{attribute 'no_check'}
FUNCTION_BLOCK IOMotor IMPLEMENTS I_ActuatorOnOff
VAR_INPUT
	ResetTrig												:	BOOL := TRUE; //Confirm error
	start													:	BOOL;
	Feed													:	BOOL;
	ProtSwitchOK											: 	FUSE;
END_VAR                 							
VAR_OUTPUT
{attribute 'displaymode':='binary'}
	Status													:	BYTE;              							
	Q_Contactor										AT  %Q* :	BOOL; //Hardware output for main contactor to start motor	
	Busy													:	BOOL;
	Error													:	BOOL;
END_VAR                 							
VAR (* IO Internal *)   							

                        	
END_VAR                 	
VAR                     	
END_VAR

(* Com Motor IO 					 		V2.2		*)
(********************************************************)

(* Protection Switch *****************************************)
	IF ResetTrig THEN reset(); END_IF

	ProtSwitchOK();

(* Enable ****************************************************)
	IF Start THEN
		switchOn();
	ELSE
		switchOff();
	END_IF
	
(* HMI status *********************************************)
	_writeStatus();
	
(********************************************************)

METHOD PROTECTED _writeStatus : BOOL
VAR_INPUT
END_VAR
	
(* HmiStatus **************************************************)
	Status.0												:= NOT Q_Contactor;
	Status.1												:= Q_Contactor;
	Status.2												:= FALSE;
	Status.3												:= FALSE;
	Status.4												:= FALSE;
	Status.5												:= Feed ;
	Status.6												:= NOT Error;
	Status.7												:= Error;

	(* Result *)
	_writeStatus											:= TRUE;
    												
(**************************************************************)
END_METHOD

METHOD enable : BOOL //Result value = successful execution of desired action 
VAR_INPUT
	IN							:	BOOL; //TRUE = Enable Pos/FWD/Up/Open/Left/Work FALSE = Opposite
END_VAR
IF in
THEN
	enable := switchOn();
ELSE
	enable := switchOff();
END_IF
END_METHOD

{attribute 'monitoring' := 'call'}
PROPERTY public inError : bool
GET
inError := Error;
END_GET
END_PROPERTY

{attribute 'monitoring' := 'call'}
PROPERTY public isBusy : bool
GET
isBusy := Busy;
END_GET
END_PROPERTY

{attribute 'monitoring' := 'call'}
PROPERTY public isOff : BOOL
GET
isOff := not Q_Contactor;
END_GET
END_PROPERTY

{attribute 'monitoring' := 'call'}
PROPERTY public isOn : BOOL
GET
isOn := Q_Contactor;
END_GET
END_PROPERTY

{attribute 'monitoring' := 'call'}
PROPERTY noFeed : BOOL
GET
noFeed := NOT Feed;
END_GET
END_PROPERTY

{attribute 'monitoring' := 'call'}
PROPERTY ok : bool
GET
ok := isBusy;
END_GET
END_PROPERTY

METHOD PUBLIC reset : bool
VAR_INPUT
END_VAR
Error									:= FALSE;
reset									:= ProtSwitchOK.reset();
END_METHOD

METHOD public switchOff : BOOL  //True if motor is switched off
VAR_INPUT
END_VAR
Start														:= FALSE;
Q_Contactor 												:= FALSE;
Busy														:= FALSE;
Error														:= NOT ProtSwitchOK.Q;
switchOff													:= TRUE;
END_METHOD

METHOD public switchOn : BOOL  //True if motor is switched on
VAR_INPUT
END_VAR
Start														:= TRUE;
Q_Contactor		 											:= ProtSwitchOK.Q AND Feed;
switchOn													:= Q_Contactor;
Busy														:= switchOn;
Error														:= NOT ProtSwitchOK.Q;
END_METHOD

END_FUNCTION_BLOCK

(* stored: Version 1.1.0.1, ProductVersion 3.1.4024.3
   POU IOMotor: Id {652201da-3ead-4c30-bab1-0ca4c35805c5}, SpecialFunc None
   Folder methods: Id {279f1738-11a0-4557-bc76-03636caa0103}
   Folder properties: Id {cdc3a8c6-d9ab-45f4-9e58-29086c8f4ca8}
   Method _writeStatus: Id {d0bf2cdc-2033-4c95-8e81-e97f00465086}
   Method enable: Id {60ee09d1-668d-4005-8dc1-fa67d9c98d07}
   Property inError: Id {008b23aa-43f0-472b-b846-0fcdb8edec46}
   Get Get: Id {85279bf0-3fcf-48a9-aa9d-ba31f3f1d85e}
   Property isBusy: Id {c381b8ab-23c8-4ba4-aa8b-2e00d6ad40c6}
   Get Get: Id {c94fec61-0c31-4feb-81d5-2e19603a09c7}
   Property isOff: Id {6a96a948-6245-40dd-970b-f1becfc150dc}
   Get Get: Id {db6bd55b-279f-4240-ac65-844e40d0f91e}
   Property isOn: Id {91a4c22d-91e5-43bb-9e58-07c31a421aba}
   Get Get: Id {a84d6782-4d21-4e27-9ea3-b4e5d4b05e92}
   Property noFeed: Id {b9e49d17-a1ba-4898-a032-f85e6c443058}
   Get Get: Id {37404ba0-2f72-440b-b7c8-d66d0c4129e1}
   Property ok: Id {564e6699-e953-4c3f-bcf7-fc181aaa237e}
   Get Get: Id {f8961047-3fab-4fa6-aa9c-a0b685ea5896}
   Method reset: Id {4671c25b-4e53-49f1-9393-a5cd4f8a4735}
   Method switchOff: Id {998f8b8e-c14f-4ee9-a6b5-29d807f55a97}
   Method switchOn: Id {aa9f363c-1580-4e6c-b4fb-8a1da6473523} *)
